FUNCTION_BLOCK FB_BoxSupplyCtrl_v1 EXTENDS FB_ObjectBase_V2
VAR_INPUT
//    Execute    :BOOL;   // True : This prog will start.
//    Abort      :BOOL;   // True : This prog will be abort.
//    Reset      :BOOL;   // True : This prog will be reset.
//    ObjectName :STRING; // Set this fb name(About it's action)

//	SupplyBTN 				:REFERENCE TO FB_Button;			//2nd machine
//	RackMotor				:REFERENCE TO FB_RackMotor_V2;
//	BoxesPusherCylinder		:REFERENCE TO FB_Cylinder;


	Cylinder				:REFERENCE TO UNI_CylinderList;
	Input 					:REFERENCE TO ST_InputTable;
	Output					:REFERENCE TO ST_OutputTable;
	fbstorageHome			: REFERENCE TO FB_StorageHoming;
	StroageRegionMode 		:E_UnitMode;
	bAddsBoxRequest 		: BOOL;
	AddBoxes_Status			:ST_AutoAddsBoxesStatus;
	AddBoxes_Ctrl			:ST_AutoAddsBoxesCommand;
	CurrentData 			: ST_SetupPara;
	
END_VAR

VAR_OUTPUT
	RackState : E_RackState;
	AxisRackMotorBTNHomeRequest	:BOOL;
//    Busy    :BOOL;        // True : This prog is running.
//    Done    :BOOL;        // True : Command has been executed.
//    Aborted :BOOL;        // True : This prog is aborted.
//    Error   :BOOL;        // True : This prog has an error.
//    ErrorID :UINT;       // Output ErrorID
//    Status  :T_MaxString; // Output this prog status by string(255bytes)
END_VAR

VAR
//    eState :E_MethodStatus_Basic;
//	uiExecutingStep : UDINT; // This var is used to been controll STATE_EXECUTING process.
//	uiResettingStep : UDINT;
//	uiAbortingStep : UDINT;
//	_Executed :BOOL; // Executing process completed.
//	_Error : BOOL; // FB has an error.
//	_ResetCompleted : BOOL; // FB resetting completed.
//	_AbortCompleted : BOOL; // FB aborting completed.
	RackMotorStationTable   : ARRAY[0..9] OF st_StationPositions;
	uiMaxRackStation :INT :=10;
	_Abort		: BOOL;
	strStatus	: STRING;
	uiResumeStep : UINT;
	ExcutingStep :E_RackState;
	trigBTN			:R_TRIG;
	trigRequest		:R_TRIG;
	tonBtnCtrl		:ton;
	tonBtnMotorCtrl	:ton;
	tonBlinkTimer :TON;
	tonBlink_Internal :TIME :=T#500MS;

END_VAR

A00_BasicUnits();
SUPER^.A10_StateControl();

ACTION A00_BasicUnits:
tonBtnCtrl(PT:=T#5S);
tonBtnMotorCtrl(PT :=T#90S);
ErrorID := 2800;
END_ACTION

METHOD GetModelState
VAR_OUTPUT
    xDone    :BOOL;
    xBusy    :BOOL;
    xError   :BOOL;
    xAborted :BOOL;
    iErrorID :UDINT;
	UniqueErrorCode : STRING;
END_VAR
xDone    := Done;
xBusy    := Busy;
xError   := Error;
xAborted := Abort;
iErrorID := ErrorID;
END_METHOD

METHOD GetName : STRING
GetName := ObjectName;
END_METHOD

METHOD PRIVATE M_Blink : BOOL
VAR_INPUT
	
END_VAR
tonBlinkTimer(IN :=NOT tonBlinkTimer.Q,
				PT := tonBlink_Internal);
IF tonBlinkTimer.Q THEN
	Output.bStorage_StackPushPbLamp := NOT Output.bStorage_StackPushPbLamp;
END_IF
END_METHOD

METHOD PRIVATE M_GetCurrentStation : BOOL
VAR
	i : UINT;
	SetPos	 :LREAL;
END_VAR

VAR_OUTPUT
	uiCurrentStation	:UINT;
END_VAR
//SetPos := THIS^.fbMotor.NcToPlc.SetPos;
SetPos := arAxisCtrl_gb[AxisNo.RackMotor].Admin.Axis.NcToPlc.SetPos;
M_RefreshStationPos();
//IF  THIS^.fbMotor.Status.Homed THEN
IF arAxisCtrl_gb[AxisNo.RackMotor].Admin.Axis.Status.Homed THEN
	FOR i:=0 TO 9 BY 1 DO 
		IF SetPos> RackMotorStationTable[i].Position-5 AND SetPos< RackMotorStationTable[i].Position+5 THEN // Range should be confirm
			uiCurrentStation :=i;
			M_GetCurrentStation :=TRUE;
			RETURN;
		END_IF
	END_FOR
	
	uiCurrentStation:=99;
	M_GetCurrentStation :=FALSE;
ELSE
	M_GetCurrentStation :=FALSE;
	uiCurrentStation:=99;
END_IF
END_METHOD

METHOD PRIVATE M_MoveToStation : BOOL
VAR_INPUT
	uiStation : UINT;
END_VAR
VAR
	bDone	:BOOL;
	uiTargetPosition	:LREAL ;
END_VAR
M_RefreshStationPos();
IF uiStation>=0 AND uiStation <10 THEN
	uiTargetPosition :=RackMotorStationTable[uiStation].Position;
	
	arAxisCtrl_gb[AxisNo.RackMotor].PosMode.Acc := CurrentData.Axes.RackMotor.HalfAuto.Acceleration;
	arAxisCtrl_gb[AxisNo.RackMotor].PosMode.Dec := CurrentData.Axes.RackMotor.HalfAuto.Deceleration;
	arAxisCtrl_gb[AxisNo.RackMotor].PosMode.Jerk := CurrentData.Axes.RackMotor.HalfAuto.Jerk;
	arAxisCtrl_gb[AxisNo.RackMotor].PosMode.Velocity := CurrentData.Axes.RackMotor.HalfAuto.Velocity;
	arAxisCtrl_gb[AxisNo.RackMotor].PosMode.Position := uiTargetPosition;
	
//	THIS^.fbMotor.MoveAbs(lrPosition	:=uiTargetPosition,
//						lrVelocity 		:=GVL.MotorCore[AxisNo.RackMotor].VCC,
//						lrAcceleration	:=GVL.MotorCore[AxisNo.RackMotor].ACC,
//						lrDeceleration	:=GVL.MotorCore[AxisNo.RackMotor].DCC,
//						lrJerk			:=GVL.MotorCore[AxisNo.RackMotor].Jerk,
//						BufferMode		:=MC_BufferMode.MC_Aborting);
	//THIS^.fbMotor.GetCmdDoneStatus(bMotionCmdDone=>bDone);
ELSE
	M_MoveToStation :=FALSE;
	RETURN;
END_IF
END_METHOD

METHOD PRIVATE M_RefreshStationPos : BOOL
VAR_INPUT
END_VAR
VAR
	i: UINT;
	position : ST_PositionTable;
END_VAR
FOR i := 0 TO 9 DO
	position :=FUN_GetPositionTableData(PositionName:='W',Index:=i,Clip:=0);
RackMotorStationTable[i].Position:= position.X_Pos;
END_FOR
	M_RefreshStationPos :=TRUE;

// todo : update position of each stations
//FOR i:=1 TO 200 BY 1 DO
//	FOR iIndex:=0 TO 9 BY 1 DO
//		IF 		
//			DAS_CoreSys.MachineControl.CurrentData.PositionTable[i].Index= iIndex AND
//			DAS_CoreSys.MachineControl.CurrentData.PositionTable[i].Zone ='W' THEN
//			RackMotorStationTable[iIndex].Position := DAS_CoreSys.MachineControl.CurrentData.PositionTable[i].X_Pos;

//			StationsPosition[iIndex]:=RackMotorStationTable[i].Position;
//		ELSE
//			M_RefreshStationPos :=FALSE;
//		END_IF
//	END_FOR
//END_FOR
END_METHOD

METHOD  M_STATE_ABORTED
VAR_INPUT
END_VAR
ERROR :=TRUE;
Busy    := FALSE;
Aborted := TRUE;
Status := strStatus;

IF NOT Execute THEN
	eSTATE:=STATE_RESETTING;
END_IF

IF Execute AND Reset THEN
	uiExecutingStep :=uiResumeStep;
	eSTATE:=STATE_EXECUTING;
END_IF
END_METHOD

METHOD  M_STATE_ABORTING
VAR_INPUT
END_VAR
CASE uiAbortingStep OF
	0 :
		uiAbortingStep:=9999;
	
	9999:	_AbortCompleted:=TRUE;
END_CASE

IF _AbortCompleted THEN	
	eSTATE :=STATE_ABORTED;
END_IF
END_METHOD

METHOD  M_STATE_DONE
VAR_INPUT
END_VAR
Busy 	:= FALSE;
Done	:=TRUE;

IF NOT Execute THEN
	eSTATE:=STATE_RESETTING;
END_IF
END_METHOD

METHOD  M_STATE_DORMANT
VAR_INPUT
END_VAR
Busy            := FALSE;
Done            := FALSE;
Aborted         := FALSE;
Error           := FALSE;
ErrorID         := 0;
Status          := '';
_ResetCompleted := FALSE;
_Error          := FALSE;
_Executed       := FALSE;
strStatus :='No Error';
uiExecutingStep :=uiResettingStep :=uiResumeStep :=0;

IF Execute THEN
	eSTATE:=STATE_EXECUTING;
END_IF
END_METHOD

METHOD  M_STATE_ERROR
VAR_INPUT
END_VAR
ERROR   :=TRUE;
Busy	:=FALSE;
Status := strStatus;
M_TurnOff();
RackState:= E_RackState.idle; // Useless so far
AxisRackMotorBTNHomeRequest :=false;
IF NOT Execute OR Reset THEN // Execute will always on , therefor Reset is only way to recovery from error	
	eSTATE:=STATE_RESETTING;
END_IF
END_METHOD

METHOD  M_STATE_EXECUTING
VAR_INPUT
END_VAR

VAR_INST
	uiTransitingStep : UINT;
	uiTargetStation :UINT :=0;
	bFreeState	  :BOOL;
END_VAR

VAR
	bMotionDone			:BOOL;
	_uiCurrentStation	:UINT;
END_VAR
Busy :=TRUE;	
//IF SupplyBTN.P_IsBTNRef THEN			//2nd machine 
//	trigBTN(CLK:= (SupplyBTN.P_ButtonState));
//END_IF //Make sure BTN is referenced otherwise exception occur

	trigBTN(CLK:= ( Input.bStorage_StackPushPb));
trigRequest(CLK :=(AddBoxes_Status.InterventionRequest AND bFreeState));

// Force state control
IF fbstorageHome.xDone THEN
	ExcutingStep := E_RackState.FeedBox;
	
ELSIF fbstorageHome.xBusy THEN
	ExcutingStep := E_RackState.ManualCtrl;
ELSIF AddBoxes_Status.Busy OR AddBoxes_Status.Done  AND NOT RackState = E_RackState.TransitingFeedBox THEN	
	ExcutingStep := E_RackState.AddBoxes;
	
ELSIF StroageRegionMode = E_UnitMode.MANUAL AND
	arAxisCtrl_gb[AxisNo.RackMotor].Admin.Axis.Status.HasJob AND
//	  rackmotor.fbMotor.Status.HasJob AND 
	  NOT (ExcutingStep = E_RackState.FeedBox)  AND 
		NOT (ExcutingStep = E_RackState.TransitingFeedBox) THEN	
			ExcutingStep := E_RackState.ManualCtrl;

ELSIF	StroageRegionMode = E_UnitMode.MANUAL AND 
		NOT Cylinder.List.fbStackPush.InRearPosition AND
//		BoxesPusherCylinder.P_IsMoving AND 
		NOT	(ExcutingStep = E_RackState.FeedBox) AND
		NOT (ExcutingStep = E_RackState.TransitingFeedBox)  THEN	
			ExcutingStep := E_RackState.ManualCtrl;

			
END_IF

RackState := ExcutingStep;

CASE ExcutingStep OF
	

	E_RackState.idle:
		;	
	E_RackState.AddBoxes:
		//Service AddBox working
		M_TurnOff();
		bFreeState:=FALSE;
		IF NOT AddBoxes_Ctrl.Execute AND NOT AddBoxes_Status.Error  THEN
        	ExcutingStep := E_RackState.Free;
    	END_IF
		
	E_RackState.ManualCtrl:
	//Stroage area in manual and Rack is moving
		M_TurnOff();
		bFreeState:=FALSE;
		IF NOT arAxisCtrl_gb[AxisNo.RackMotor].Admin.Axis.Status.HasJob AND Cylinder.List.fbStackPush.InRearPosition THEN
            ExcutingStep := E_RackState.Free;
        END_IF
		
	E_RackState.FeedBox:
	// FeedBox mode , 
		M_Blink();
		bFreeState:=FALSE;
		AxisRackMotorBTNHomeRequest :=false;
			IF	trigBTN.Q THEN				
				ExcutingStep :=E_RackState.TransitingFree;	
			END_IF
			
	E_RackState.Free:
	// Rack is free , User is allow to ask to suply box by push the suplyBTN
		M_TurnOn();
		bFreeState:=TRUE;
			 IF trigBTN.Q OR trigRequest.Q THEN
				 uiTransitingStep:=0;
				 ExcutingStep := E_RackState.TransitingFeedBox;
			 END_IF

	E_RackState.TransitingFree:
			 IF NOT AddBoxes_Status.InterventionRequest THEN
				 ExcutingStep :=E_RackState.Free;	
			 END_IF
		
	E_RackState.TransitingFeedBox:
	//Transition step , from Free to FeedBox
		//M_Blink();
		M_TurnOff();
		bFreeState:=FALSE;
		AxisRackMotorBTNHomeRequest :=TRUE;
		// todo : if transition step needs different indication of BTN behavior?
		CASE uiTransitingStep OF
		0:
			tonBtnCtrl.IN	:=FALSE;
			tonBtnMotorCtrl.IN :=FALSE;
			uiTransitingStep:=5;
			M_GetCurrentStation(uiCurrentStation =>_uiCurrentStation);
			IF uiTargetStation = _uiCurrentStation THEN
				uiTransitingStep :=30;
			END_IF
			
		5:	//Move cylinder back
			tonBtnCtrl.IN:=TRUE;			
			Cylinder.List.fbStackPush.M_Retract();
			IF Cylinder.List.fbStackPush.InRearPosition AND NOT arAxisCtrl_gb[AxisNo.RackMotor].Admin.Axis.Status.HasJob THEN 
				tonBtnCtrl.IN :=FALSE;
				uiTransitingStep :=10;
			END_IF
			IF tonBtnCtrl.Q THEN
				_Error:= TRUE;
				StrStatus :='Cylinder MoveBackward timeout';
			END_IF
		10:	// Rackmotor move to station 0
			tonBtnMotorCtrl.IN :=TRUE;
			M_MoveToStation(uiTargetStation);
			IF arAxisCtrl_gb[AxisNo.RackMotor].Admin.Axis.Status.HasJob THEN
			uiTransitingStep :=20;
			END_IF
			IF tonBtnMotorCtrl.Q THEN
				_Error :=TRUE;
				StrStatus :='RackMotor MoveToStation timeout';
			END_IF
		20:	// check currentstation 
			tonBtnMotorCtrl.IN :=TRUE;
//			bMotionDone :=rackmotor.fbMotor.Status.InTargetPosition;
			bMotionDone :=arAxisCtrl_gb[AxisNo.RackMotor].Admin.Axis.Status.InTargetPosition;
			M_GetCurrentStation(uiCurrentStation =>_uiCurrentStation);
			IF bMotionDone  AND uiTargetStation = _uiCurrentStation THEN
				tonBtnMotorCtrl.IN :=FALSE;
				uiTransitingStep :=30;
			END_IF
			IF tonBtnMotorCtrl.Q THEN
				_Error :=TRUE;
				StrStatus :='RackMotor currentStation timeout';
			END_IF
		30:
			ExcutingStep := E_RackState.FeedBox;
			AxisRackMotorBTNHomeRequest :=FALSE;
		END_CASE
		


END_CASE
	
IF NOT Execute THEN
	eState:=STATE_RESETTING;
END_IF
IF _Error THEN
	eState:=STATE_ERROR;
END_IF
IF _Abort THEN
	eSTATE:=STATE_ABORTING;
END_IF
IF _Executed THEN
	eSTATE:=STATE_Done;
END_IF
END_METHOD

METHOD  M_STATE_RESETTING
VAR_INPUT
END_VAR
Error :=FALSE;
Done :=FALSE;
Busy := FALSE;
AxisRackMotorBTNHomeRequest :=FALSE;
tonBtnCtrl.IN := FALSE;
tonBtnMotorCtrl.IN := FALSE;
M_TurnOff();
CASE uiResettingStep OF
	
	0:
		uiResettingStep:=9999;


	9999:
		_ResetCompleted:=TRUE;
END_CASE
IF _ResetCompleted THEN
	eSTATE:=STATE_DORMANT;
END_IF
END_METHOD

METHOD PRIVATE M_TurnOff : BOOL
VAR_INPUT
END_VAR
Output.bStorage_StackPushPbLamp := false;
END_METHOD

METHOD PRIVATE M_TurnOn : BOOL
VAR_INPUT
END_VAR
Output.bStorage_StackPushPbLamp := true;
END_METHOD

END_FUNCTION_BLOCK

(* stored: Version 1.1.0.1, ProductVersion 3.1.4024.13
   POU FB_BoxSupplyCtrl_v1: Id {3b39c6b2-63b1-4bd4-bc54-04a970e26fef}, SpecialFunc None
   Folder Private: Id {48775554-6c83-4429-98ff-e11c4778753b}
   Folder STATE: Id {0599fb81-bfb1-4dfb-874d-ae888c88eba6}
   Action A00_BasicUnits: Id {cec0843e-2423-44ee-b8ef-4e12bf139a55}
   Method GetModelState: Id {4267a49d-0356-49cd-b4a8-19cde37ac0cb}
   Method GetName: Id {31a1fe00-1ad2-41e2-b58c-7efc37a3b636}
   Method M_Blink: Id {64b9d6b9-97dd-4747-b150-b278e8f442ce}
   Method M_GetCurrentStation: Id {56b38c74-8a8d-4896-af92-c1e7e9ddb7b4}
   Method M_MoveToStation: Id {e7037cb5-7713-474a-8085-e388588abd5f}
   Method M_RefreshStationPos: Id {3a97fa84-8273-492c-b394-febc28ec994a}
   Method M_STATE_ABORTED: Id {0ed5a138-dcc6-4a55-84b6-153d51b51b99}
   Method M_STATE_ABORTING: Id {62848b8d-0669-432d-a705-960fb43b2765}
   Method M_STATE_DONE: Id {97b1f544-094d-4d3a-b39e-883a332de507}
   Method M_STATE_DORMANT: Id {a84f19e5-bab9-4e27-a46c-6ad713e5640e}
   Method M_STATE_ERROR: Id {25173218-b8b4-4514-bc59-3f87f416bb0b}
   Method M_STATE_EXECUTING: Id {1f97a79b-4cf9-4894-a872-728d778ffa16}
   Method M_STATE_RESETTING: Id {63a41575-6e45-4e09-be92-e0d647b78c57}
   Method M_TurnOff: Id {6be90b55-1270-4dc5-8ca9-0a07ecd719d0}
   Method M_TurnOn: Id {c132d2ba-6958-4613-8a2c-e5a295bb195f} *)
